ABB RobotStudio station: PracticaEntregable2AvanzadaEstacionDePartida(1).rspag

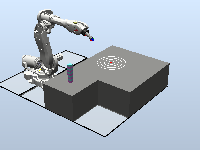
--- station ---
Station Practica3Avanzada_EstacionDePartida (saved by RobotStudio 6.6.7701.1025)
Controller Sistema6
  mechanical unit ROB_1: IRB6640_180_255__04, 6 joints, base frame (0, 0, 0) mm
Layout (positions relative to the parent item):
  - Ventosa [mechanism] at (1635.71, 0, 1955) mm, rotated rx 180 ry 60 rz 180 deg
      TCP Ventosa at (0, 0, 200) mm
      links: PiezaVentosa
  - IRB6640_180_255__04 [mechanism, from Robots\IRB6640_180_255_G_04.rslib] at (0, 0, 0) mm; joint values [0, 0, 0, 0, 0.5236, 0] (rad or m)
  - MesaTrabajoParte1 [part]
  - MesaTrabajoParte0 [part]
  - CI_VentosaVacuostato [smart component]
      signals: DI ActivaVentosa, DO Vacuostato
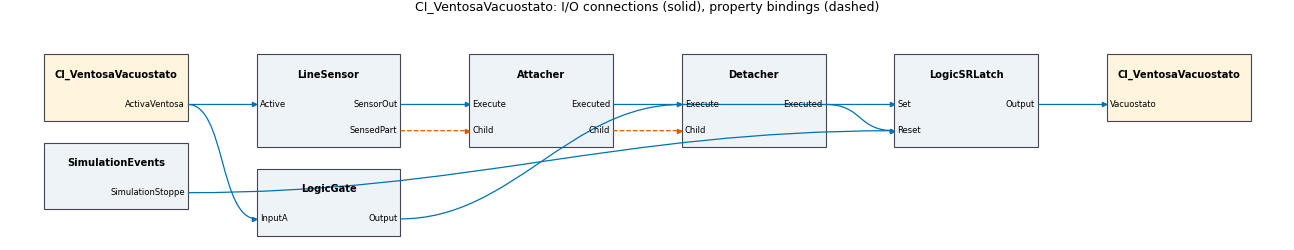
      connections:
        CI_VentosaVacuostato.ActivaVentosa -> LineSensor.Active
        LineSensor.SensorOut -> Attacher.Execute
        Attacher.Executed -> LogicSRLatch.Set
        LogicSRLatch.Output -> CI_VentosaVacuostato.Vacuostato
        Detacher.Executed -> LogicSRLatch.Reset
        SimulationEvents.SimulationStopped -> LogicSRLatch.Reset
        CI_VentosaVacuostato.ActivaVentosa -> LogicGate.InputA
        LogicGate.Output -> Detacher.Execute
        LineSensor.SensedPart => Attacher.Child
        Attacher.Child => Detacher.Child
    - LineSensor [smart component, from Components\LineSensor.rslib] at (1808.91, 0, 1855) mm, rotated rx 180 ry 60 rz 180 deg
        properties: Start=[0 0 -0.002]; End=[0 0 0.02]; Radius=0.002; SensedPart=(none); SensedPoint=[1.50000012207031 0.500000030517578 0.85]
      - _sensorPart_ [part]
    - SimulationEvents [smart component, from Components\SimulationEvents.rslib]
    - LogicSRLatch [smart component, from Components\LogicSRLatch.rslib]
    - Attacher [smart component, from Components\Attacher.rslib]
        properties: Parent=Ventosa; Flange=0; Child=(none); Mount=false; Offset=[0 0 0]; Orientation=[0 0 0]
    - Detacher [smart component, from Components\Detacher.rslib]
        properties: Child=(none); KeepPosition=true
    - LogicGate [smart component, from Components\LogicGate.rslib]
        properties: Operator=NOT; Delay=0.1
  - MesaTrabajoParte2 [part] at (0, 1000, 0) mm
  - MesaTrabajoParte3 [part] at (1000, 0, 0) mm
  - MesaTrabajoParte4 [part] at (1000, 1000, 0) mm
  - Pieza1 [part]
  - Pieza2 [part]
  - Pieza3 [part]
  - Pieza4 [part]
  - Pieza5 [part]
  - CircunferenciaR200 [part]
  - CircunferenciaR100 [part]
  - CircunferenciaR300 [part]
  - CircunferenciaR400 [part]
  - Pieza6 [part]
  - Pieza7 [part]
  - Pieza8 [part]
  - Pieza9 [part]
  - Pieza10 [part]
Attachment: Ventosa is attached to IRB6640_180_255__04 / Link6
Attachment: LineSensor is attached to Ventosa / PiezaVentosa
Station logic (signal -> signal, property => property):
  CI_VentosaVacuostato.Vacuostato -> Sistema6.ED_PiezaCogida
  Sistema6.SD_ActivaVentosa -> CI_VentosaVacuostato.ActivaVentosa

--- Backups/Sistema6/RAPID/TASK1/PROGMOD/CalibData.mod ---
MODULE CalibData
	PERS tooldata Ventosa:=[TRUE,[[0,0,200],[1,0,0,0]],[1,[0,0,125],[1,0,0,0],0.002,0.002,0.0013]];
ENDMODULE

--- Backups/Sistema6/RAPID/TASK1/PROGMOD/Module1.mod ---
MODULE Module1
    CONST robtarget pBaseOrigen:=[[1500,-500,750],[0,0,1,0],[0,0,0,0],[9E+09,9E+09,9E+09,9E+09,9E+09,9E+09]];
    CONST robtarget pCentroDestino:=[[1700,1000,750],[0,0,1,0],[0,0,0,0],[9E+09,9E+09,9E+09,9E+09,9E+09,9E+09]];
    CONST robtarget pReposo:=[[1808.910161514,0,1855],[0.5,0,0.866025404,0],[0,0,0,0],[9E+09,9E+09,9E+09,9E+09,9E+09,9E+09]];

ENDMODULE

--- Backups/Sistema6/RAPID/TASK1/SYSMOD/LINKEDM.sys ---
%%%
  VERSION:1
  LANGUAGE:ENGLISH
%%%

MODULE LINKEDM (SYSMODULE)

! FOLLOWER
!     Name of electronically linked follower axis used by operator at teach pendent.
      PERS string l_f_axis_name{5}       :=  ["",  "", "", "", ""];

!     Name of the mechanical unit for follower axis.
      PERS string l_f_mecunt_n{5}  :=  ["", "", "", "", ""];

!     Linked follower axis number in the mechanical unit (first axis in mech. unit is number 1).
      PERS num l_f_axis_no{5}      :=  [0,          0,   0,  0,  0];

! MASTER
!     Name of the mechanical unit for linked master axis.
      PERS string l_m_mecunt_n{5} :=  ["", "", "", "", ""];

!     Linked master axis number in the mechanical unit (first axis in mech. unit is number 1).
!     See axis number table in documentation for different master mechanical units.
      PERS num l_m_axis_no{5}     :=  [0,  0,  0,  0,  0];

! POSITION OFFSET
!     The increase of the allowed offset position between the master and follower
!     positions, used when starting AUTO mode. As soon as the offset is decreased
!     the old configurated parameter is used.
!     Example: 3 => the configurated value of allowed offset is increased 3 times.
      PERS num offset_ratio{5}       :=  [10,  10,   10,  10,  10];

! SPEED RATIO
!     Speed_ratio used in AUTO and JOG modes [ very_slow   slow    normal    fast]
!     Value 1 = max allowed manual speed.
      CONST num speed_ratio {20}      := [0.01, 0.01, 0.01, 0.01, 0.01,
                                          0.05, 0.05, 0.05, 0.05, 0.05,
                                          0.20, 0.20, 0.20, 0.20, 0.20,
                                          1.00, 1.00, 1.00, 1.00, 1.00];

! STEP SIZE
!     Displacement position used in JOG mode for each activation of positive or
!     negative movement.                  [very_short    short   normal   long]
!     Unit degees or meter.
      CONST num displacement {20}     := [0.001, 0.001, 0.001, 0.001, 0.001,
                                          0.005, 0.005, 0.005, 0.005, 0.005,
                                          0.020, 0.020, 0.020, 0.020, 0.020,
                                          0.100, 0.100, 0.100, 0.100, 0.100];


!-------------------------------------------------------------
 PROC Linked_m ()
      Linked_m_exe ;
 ENDPROC
ENDMODULE

--- Backups/Sistema6/SYSPAR/EIO.cfg ---
EIO:CFG_1.0:6:1::
#
INDUSTRIAL_NETWORK:

      -Name "DeviceNet" -Label "DeviceNet Master/Slave Network" -Address "2"
#
DEVICENET_DEVICE:

      -Name "MiDeviceNet" -Label "MiDeviceNet"
#
DEVICENET_INTERNAL_DEVICE:

      -Name "DN_Internal_Device" -VendorName "ABB Robotics"\
      -ProductName "DeviceNet Internal Slave Device"
#
EIO_SIGNAL:

      -Name "ED_PiezaCogida" -SignalType "DI" -Device "MiDeviceNet"\
      -Label "ED_PiezaCogida" -DeviceMap "0" -Access "All"

      -Name "SD_ActivaVentosa" -SignalType "DO" -Device "MiDeviceNet"\
      -Label "SD_ActivaVentosa" -DeviceMap "0" -Access "All"
